(* IEC 61131-3 sources: AXOpen/src/components.siem.communication/app/SystemConstants, 2 files *)

(* ---- plc_line_IoAddresses.st ---- *)
CONFIGURATION IoAddresses
    VAR_GLOBAL

        // Module et200sp/CpPtp
        et200sp_CpPtp_Input AT %IB0 : et200sp_CpPtp_Input_Layout;
    END_VAR
END_CONFIGURATION

TYPE
    et200sp_CpPtp_Input_Layout : STRUCT
        Signals_0 AT %B0 : BYTE;
        Signals_1 AT %B1 : BYTE;
        Signals_2 AT %B2 : BYTE;
        Signals_3 AT %B3 : BYTE;
        Signals_4 AT %B4 : BYTE;
        Signals_5 AT %B5 : BYTE;
        Signals_6 AT %B6 : BYTE;
        Signals_7 AT %B7 : BYTE;
    END_STRUCT;
END_TYPE

(* ---- plc_line_HwIdentifiers.st ---- *)
CONFIGURATION HardwareIDs
    VAR_GLOBAL CONSTANT
        et200sp_HwID : UINT := UINT#258;
        et200sp_CpPtp_CM_PtP_V2_0_HwID : UINT := UINT#264;
        et200sp_Rack_HwID : UINT := UINT#261;
        et200sp_Server_module_V1_1_Server_module_V1_1_0_bytes_HwID : UINT := UINT#263;
        et200sp_et200sp_HwID : UINT := UINT#262;
        et200sp_et200sp_IM_155_6_PN_ST_V4_2_HwID : UINT := UINT#265;
        et200sp_et200sp_Port_1_HwID : UINT := UINT#259;
        et200sp_et200sp_Port_2_HwID : UINT := UINT#260;
        et200sp_et200sp_profinet_HwID : UINT := UINT#257;
        plc_line_HwID : UINT := UINT#32;
        plc_line_Rail_0_HwID : UINT := UINT#266;
        plc_line_plc_line_HwID : UINT := UINT#48;
        plc_line_plc_line_CPU_display_1_HwID : UINT := UINT#54;
        plc_line_plc_line_Card_reader_writer_1_HwID : UINT := UINT#51;
        plc_line_plc_line_DP_interface_1_HwID : UINT := UINT#60;
        plc_line_plc_line_OPC_UA_1_HwID : UINT := UINT#117;
        plc_line_plc_line_PROFINET_interface_1_HwID : UINT := UINT#64;
        plc_line_plc_line_PROFINET_interface_1_Port_1_HwID : UINT := UINT#65;
        plc_line_plc_line_PROFINET_interface_1_Port_2_HwID : UINT := UINT#66;
        plc_line_plc_line_PROFINET_interface_2_HwID : UINT := UINT#72;
        plc_line_plc_line_PROFINET_interface_2_Port_3_HwID : UINT := UINT#73;
        plc_line_plc_line_Virtual_communication_interface_HwID : UINT := UINT#135;
        profinet_plc_line_HwID : UINT := UINT#256;

    END_VAR
END_CONFIGURATION
